// SIMATIC S7-200 project (STEP 7-Micro/WIN), CPU 226 REL 02.00

SYMBOL_TABLE I
                 ?0_40_0  // 镀镍反应池加碱压力开关71
                 ?0_40_0  // 配碱切断阀
                 ?0_40_0  // 配酸切断阀
PDT101           AIW0     // PDT101（镀镍废水过滤器）
AIT101           AIW2     // AIT101PH（镀镍废水调节池PH）
AIT102           AIW4     // AIT102PH（镀镍反应池1#PH）
AIT103           AIW6     // AIT103PH（镀镍反应池2#PH）
FIQ100           AIW8     // FIQ100（镀镍进水总计量）
LT401            AIW10    // 酸液位LT401
LT402            AIW12    // 碱液位LT402
                 AIW14    // 可燃气体报警（未找到）
AIT106           AIW16    // AIT106（NF进水CI）
LS101A           I0.0     // 1#中继池液位高
LS101B           I0.1     // 1#中继池液位高高
M103C_RUN        I0.3     // 反应池搅拌机A运行反馈
M101A_RUN        I0.4     // 镀镍1#中继池提升泵A运行反馈
M101B_RUN        I0.5     // 镀镍1#中继池提升泵B运行反馈
M103D_RUN        I0.6     // 反应池搅拌机B运行反馈
M103C_OVER       I0.7     // 反应池搅拌机A过载
M101A_OVER       I1.0     // 镀镍1#中继池泵A运行过载
M101B_OVER       I1.1     // 镀镍1#中继池泵B运行过载
M103D_OVER       I1.2     // 反应池搅拌机B过载
DUNIE2_H         I1.3     // 镀镍2#中继池液位高
YJC_1A_RUN       I1.4     // 1#应急池提升泵A运行状态14
YJC_1B_RUN       I1.5     // 1#应急池提升泵B运行状态15
YJC_2A_RUN       I1.6     // 2#应急池提升泵A运行状态16
YJC_2B_RUN       I1.7     // 2#应急池提升泵B运行状态17
M402A_RUN        I2.0     // 碱泵A运行反馈M401C
M402B_RUN        I2.1     // 碱泵B运行反馈M401D
M401A_RUN        I2.2     // 酸泵A运行反馈M401A
M401B_RUN        I2.3     // 酸泵B运行反馈M401B
YJC_1A_OVER      I2.4     // 1#应急池提升泵A过载状态24
YJC_1B_OVER      I2.5     // 1#应急池提升泵B过载状态25
YJC_1L           I2.6     // 1#应急池液位计低2.6
YJC_1H           I2.7     // 1#应急池液位计高2.7
YJC_2L           I3.0     // 2#应急池液位计低3.0
YJC_2H           I3.1     // 2#应急池液位计高3.1
JIAN_YEWEI       I3.2     // 镀镍反应池加碱液位计no
DUNIE2_L         I3.3     // 镀镍2#中继池液位低
YJC_2A_OVER      I3.4     // 2#应急池提升泵A过载状态34
YJC_2B_OVER      I3.5     // 2#应急池提升泵B过载状态35
M402A_OVER       I3.6     // 碱泵A过载M401C
M402B_OVER       I3.7     // 碱泵B过载M401D
M401A_OVER       I4.0     // 酸泵A过载M401A
M401B_OVER       I4.1     // 酸泵B过载M401B
JBJ_QPJ_RUN      I5.0     // 配消泡剂搅拌机运行状态60
M410_OVER        I5.1     // 配PAC搅拌机过载状态61
M103E_OVER       I5.2     // 镀镍反应池加碱过载状态62
M401C_OVER       I5.3     // 配酸搅拌机过载状态63
M402C_OVER       I5.4     // 配碱搅拌机过载状态64
JBJ_QPJ_OVER     I5.5     // 配消泡剂搅拌机过载状态65
M410_RUN         I6.4     // 配PAC搅拌机运行状态54
M103E_RUN        I6.5     // 镀镍反应池加碱运行状态55
M401C_RUN        I6.6     // 配酸搅拌机运行状态56
M402C_RUN        I6.7     // 配碱搅拌机运行状态57
UF_YW_H          I7.0     // 超滤中间水箱液位高
SV106A_RUN       I7.1     // 过滤器切断阀1运行反馈
SV106B_RUN       I7.2     // 过滤器切断阀2运行反馈
SV106C_RUN       I7.3     // 过滤器切断阀3运行反馈
DUNIE_A_RUN      I7.4     // 镀镍2#中继池提升泵B运行
DUNIE_B_RUN      I7.5     // 镀镍2#中继池提升泵A运行
DUNIE_A_OVER     I7.6     // 镀镍2#中继池提升泵B过载
DUNIE_B_OVER     I7.7     // 镀镍2#中继池提升泵A过载
M103A_RUN        I8.2     // 镀镍调节池提升泵A运行状态82
M103B_RUN        I8.3     // 镀镍调节池提升泵B运行状态83
M103A_OVER       I8.4     // 镀镍调节池提升泵A过载状态84
M103B_OVER       I8.5     // 镀镍调节池提升泵B过载状态85
TJCYW_L          I8.6     // 镀镍调节池液位计(起泵位)8.6
TJCYW_H          I8.7     // 镀镍调节池液位计(低保护)8.7
                          // 集水井液位计no
END_SYMBOL_TABLE

SYMBOL_TABLE Q
                 ?0_40_0  // 集水井提升泵A运行
                 ?0_40_0  // 集水井提升泵B运行
M101A            Q0.0     // 镀镍1#中继池提升泵A运行00
M101B            Q0.1     // 镀镍1#中继池提升泵B运行01
DUNIE_A          Q0.2     // 镀镍2#中继池提升泵B运行7#
DUNIE_B          Q0.3     // 镀镍2#中继池提升泵A运行7#
YJC_PUMPA        Q0.4     // 应急池提升泵A
YJC_PUMPB        Q0.5     // 应急池提升泵B
YJC_PUMPC        Q0.6     // 应急池提升泵C
YJC_PUMPD        Q0.7     // 应急池提升泵D
M402A            Q1.0     // 酸提升泵A
M402B            Q1.1     // 酸提升泵B
M401A            Q1.2     // 碱提升泵A
M401B            Q1.3     // 碱提升泵B
M410             Q2.1     // 配PAC搅拌机运行54
M103E            Q2.2     // 镀镍反应池加碱运行22
M401C            Q2.3     // 配酸搅拌机运行23
M402C            Q2.4     // 配碱搅拌机运行57
JBJ_QPJ          Q2.5     // 配消泡剂搅拌机运行60
LV401            Q2.6     // 酸加水阀门26
LV402            Q2.7     // 碱加水阀门27
M103A            Q3.0     // 镀镍调节池池提升泵A
M103B            Q3.1     // 镀镍调节池池提升泵B
M103C            Q3.2     // 反应池搅拌机Ano
M103D            Q3.3     // 反应池搅拌机Bno
SV106A           Q3.4     // 过滤器切断阀1no
SV106B           Q3.5     // 过滤器切断阀2no
SV106C           Q3.6     // 过滤器切断阀3no
END_SYMBOL_TABLE

SYMBOL_TABLE M
AUTO             M0.0     // 手/自动
                 M0.2     // 中间水箱液位高标志
                 M0.3     // 调节池泵启动条件
                 M0.4     // M401AB
                 M0.5     // M402AB
SV106_ID         M0.7     // 置过滤器截断阀运行标志位
                 M1.0     // 镀镍2#中继池启动条件
                 M1.1     // 1#应急池提升泵启动条件
                 M1.2     // 2#应急池提升泵启动条件
                 M1.3     // 镀镍1#中继池启动条件
FYC_ALARM        M1.4     // 反应池PH报警
ALARM_EN         M2.0     // 报警
TJC_ALARM        M2.1     // 调节池PH报警
TJC_ALARM_R      M2.2     // 调节池PH报警复位
                 M10.0    // AIT101报警
                 M10.1    // PDT101报警
                 M10.2    // AIT102报警
                 M10.3    // AIT103报警
                 M10.4    // FE101报警
                 M10.5    // 可燃气体报警
                 M10.6    // 酸液位报警
                 M10.7    // 碱液位报警
                 M11.0    // AIT106报警
M112             M11.2    // 镀镍2#中继池提升泵A在线
M113             M11.3    // 镀镍2#中继池提升泵B在线
M156             M15.6    // 酸单次配药
M157             M15.7    // 碱单次配药
M160             M16.0    // 反应池PH压力联锁允许
M161             M16.1    // 反应池PH液位联锁允许
M162             M16.2    // 反应池PH自动控制
M163             M16.3    // 调节池提升泵允许PH控制
M164             M16.4    // 调节池PH报警
M165             M16.5    // 过滤器压力报警允许
M166             M16.6    // 调节池液位允许提升泵启动综合状态
M167             M16.7    // 酸自动配药
M170             M17.0    // 碱自动配药
M171             M17.1    // 2#应急池提升泵液位联锁允许
M172             M17.2    // 1#应急池提升泵液位联锁允许
M173             M17.3    // 镀镍调节池提升泵液位联锁允许
M174             M17.4    // 镀镍2#中继池提升泵液位联锁允许
M175             M17.5    // 镀镍1#中继池提升泵液位联锁允许
M176             M17.6    // 镀镍反应池搅拌机联锁允许
M182             M18.2    // 集水井提升泵B在线
M183             M18.3    // 集水井提升泵A在线
M184             M18.4    // 配消泡剂搅拌机在线
M185             M18.5    // 配PAC搅拌机在线
M186             M18.6    // 配碱搅拌机在线
M187             M18.7    // 配酸搅拌机在线
M190             M19.0    // 碱输送泵A在线
M191             M19.1    // 碱输送泵B在线
M192             M19.2    // 酸输送泵A在线
M193             M19.3    // 酸输送泵B在线
M194             M19.4    // 2#应急池提升泵B在线
M195             M19.5    // 2#应急池提升泵A在线
M196             M19.6    // 1#应急池提升泵B在线
M197             M19.7    // 1#应急池提升泵A在线
M200             M20.0    // 镀镍反应池加碱在线
M201             M20.1    // 镀镍反应池搅拌机A在线
M202             M20.2    // 镀镍反应池搅拌机B在线
M203             M20.3    // 镀镍调节池提升泵A在线
M204             M20.4    // 镀镍调节池提升泵B在线
M205             M20.5    // 镀镍1#中继池提升泵A在线
M206             M20.6    // 镀镍1#中继池提升泵B在线
M211             M21.1    // 过滤器切断阀1在线
M212             M21.2    // 过滤器切断阀2在线
M213             M21.3    // 过滤器切断阀3在线
M214             M21.4    // 镀镍反应池加碱压力保护允许
M215             M21.5    // 过滤器切断阀
END_SYMBOL_TABLE

SYMBOL_TABLE TC
                 T37      // AB切换定时
                 T38      // AB定时辅助
                 T254     // 报警延时
END_SYMBOL_TABLE

SYMBOL_TABLE V
                 VD300    // AIT101最大设定值
                 VD304    // AIT101最小设定值
                 VD308    // PDT101最大设定值
                 VD312    // PDT101最小设定值
                 VD316    // AIT102最大设定值
                 VD320    // AIT102最小设定值
                 VD324    // AIT103最大设定值
                 VD328    // AIT103最小设定值
                 VD332    // FE101最大设定值
                 VD336    // FE101最小设定值
                 VD340    // 可燃气体报警最大设定值
                 VD344    // 可燃气体报警最小设定值
                 VD348    // 酸液位最大设定值
                 VD352    // 酸液位最小设定值
                 VD356    // 碱液位最大设定值
                 VD360    // 碱液位最小设定值
                 VD364    // AIT106最大设定值
                 VD368    // AIT106最小设定值
PDT              VW0      // PDT101
TJC_PH           VW2      // AIT101
FYC_PH1          VW4      // AIT102
FYC_PH2          VW6      // AIT103
FE101            VW8      // FE101
SUAN_YW          VW10     // 酸液位
JIAN_YW          VW12     // 碱液位
                 VW14     // 可燃气体报警
                 VW16     // AIT106镀镍纳虑进水电导率
S125             VW18     // 调节池PH报警设定值高8.0
S126             VW20     // 反应池PH1低限设定值6.0
S127             VW22     // 反应池PH1高限设定值8.0
S128             VW24     // 酸加水高度设定值1-30
S129             VW26     // 酸加酸高度设定值2-60
S130             VW28     // 酸加水高度设定值3-100
S131             VW30     // 碱加水高度设定值1
S132             VW32     // 碱加碱高度设定值2
S133             VW34     // 碱加水高度设定值3
                 VW36     // 调节池PH报警设定值低
                 VW42     // PDT101最大设定值10
TIME1            VW100    // 定时切换时间(分钟)30
END_SYMBOL_TABLE

ORGANIZATION_BLOCK MAIN:OB1
TITLE=PROGRAM COMMENTS
BEGIN
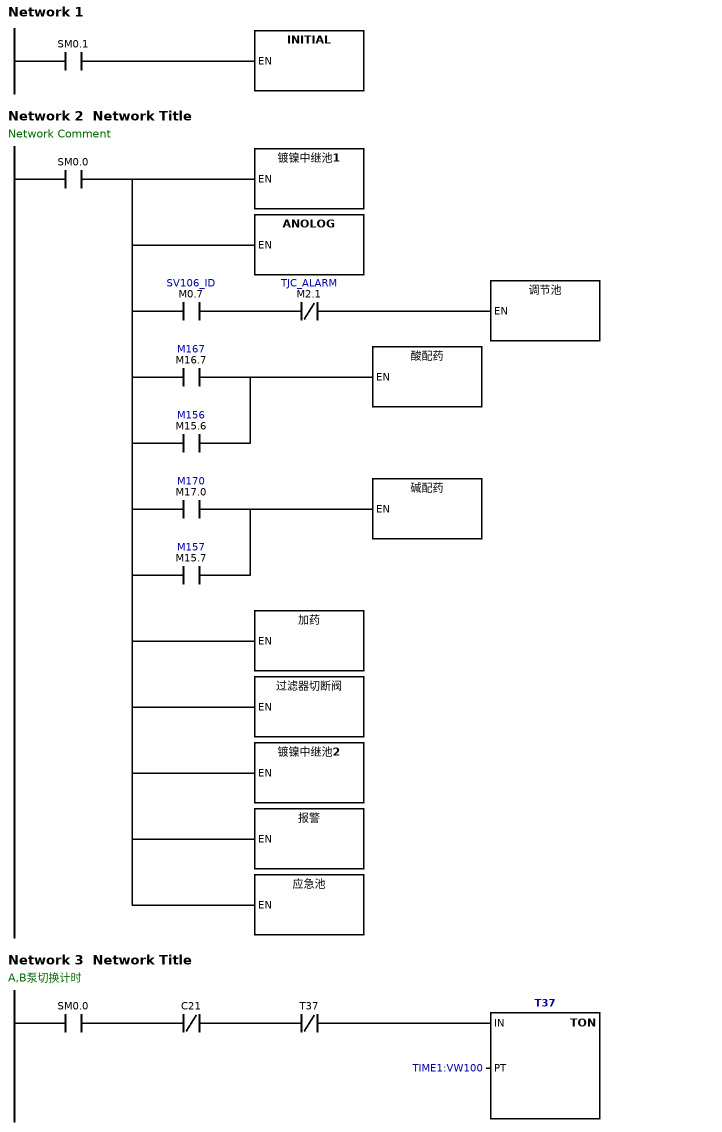
Network 1
// (network saved uncompiled; LAD cells follow)
// row 0: c0 -| |- SM0.1  c1 --  c2 [INITIAL EN:=power@row0]
Network 2 // Network Title
// Network Comment
LD     SM0.0
LPS
CALL   镀镍中继池1:SBR0
CALL   ANOLOG:SBR4
A      SV106_ID:M0.7
AN     TJC_ALARM:M2.1
CALL   调节池:SBR3
LRD
LD     M167:M16.7
O      M156:M15.6
ALD
CALL   酸配药:SBR5
LRD
LD     M170:M17.0
O      M157:M15.7
ALD
CALL   碱配药:SBR6
LPP
CALL   加药:SBR2
CALL   过滤器切断阀:SBR9
CALL   镀镍中继池2:SBR7
CALL   报警:SBR8
CALL   应急池:SBR1
Network 3 // Network Title
// A,B泵切换计时
LD     SM0.0
AN     C21
AN     T37
TON    T37, TIME1:VW100
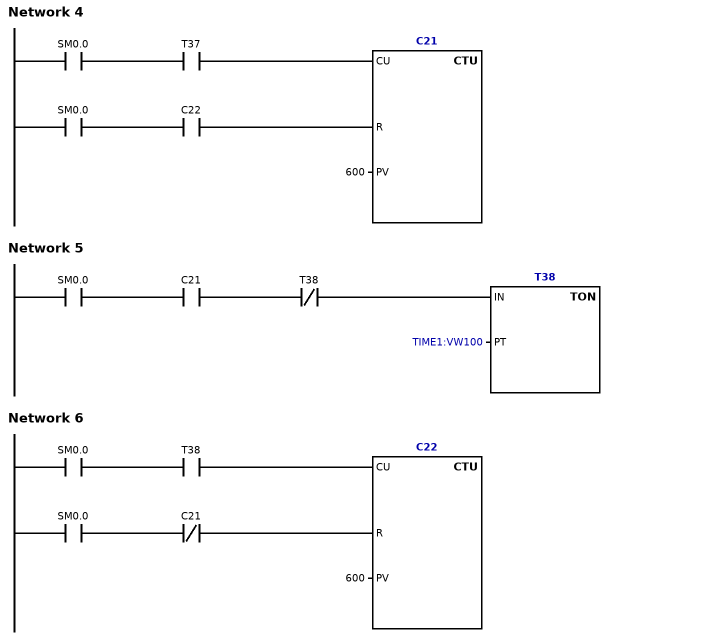
Network 4
LD     SM0.0
A      T37
LD     SM0.0
A      C22
CTU    C21, 600
Network 5
LD     SM0.0
A      C21
AN     T38
TON    T38, TIME1:VW100
Network 6
LD     SM0.0
A      T38
LD     SM0.0
AN     C21
CTU    C22, 600
END_ORGANIZATION_BLOCK

SUBROUTINE_BLOCK 镀镍中继池1:SBR0
TITLE=1#中继池
BEGIN
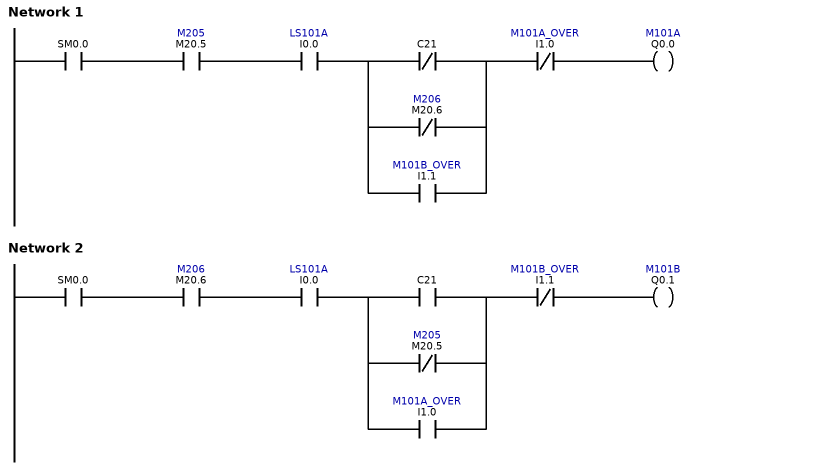
Network 1
LD     SM0.0
A      M205:M20.5
A      LS101A:I0.0
LDN    C21
ON     M206:M20.6
O      M101B_OVER:I1.1
ALD
AN     M101A_OVER:I1.0
=      M101A:Q0.0
Network 2
LD     SM0.0
A      M206:M20.6
A      LS101A:I0.0
LD     C21
ON     M205:M20.5
O      M101A_OVER:I1.0
ALD
AN     M101B_OVER:I1.1
=      M101B:Q0.1
END_SUBROUTINE_BLOCK

SUBROUTINE_BLOCK 应急池:SBR1
TITLE=子程序注释
BEGIN
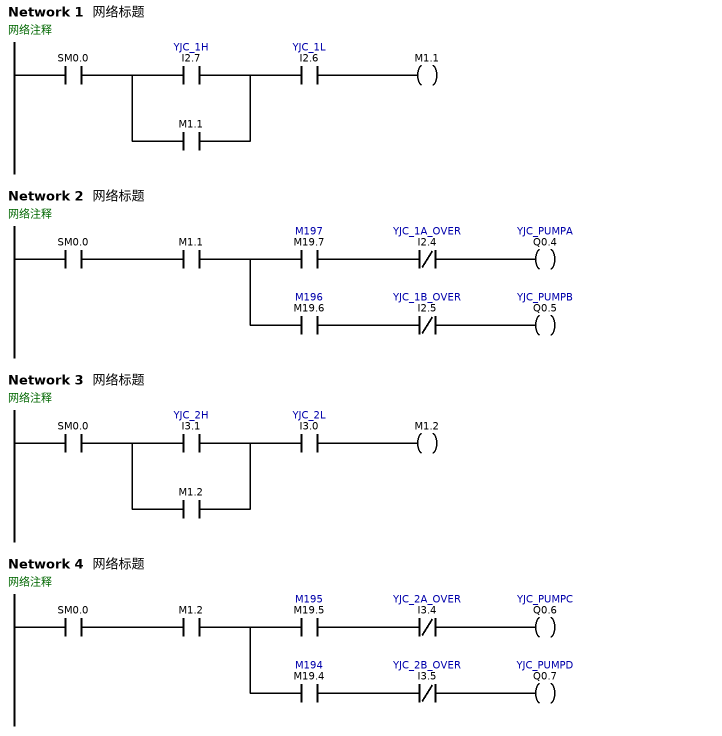
Network 1 // 网络标题
// 网络注释
LD     SM0.0
LD     YJC_1H:I2.7
O      M1.1
ALD
A      YJC_1L:I2.6
=      M1.1
Network 2 // 网络标题
// 网络注释
LD     SM0.0
A      M1.1
LPS
A      M197:M19.7
AN     YJC_1A_OVER:I2.4
=      YJC_PUMPA:Q0.4
LPP
A      M196:M19.6
AN     YJC_1B_OVER:I2.5
=      YJC_PUMPB:Q0.5
Network 3 // 网络标题
// 网络注释
LD     SM0.0
LD     YJC_2H:I3.1
O      M1.2
ALD
A      YJC_2L:I3.0
=      M1.2
Network 4 // 网络标题
// 网络注释
LD     SM0.0
A      M1.2
LPS
A      M195:M19.5
AN     YJC_2A_OVER:I3.4
=      YJC_PUMPC:Q0.6
LPP
A      M194:M19.4
AN     YJC_2B_OVER:I3.5
=      YJC_PUMPD:Q0.7
END_SUBROUTINE_BLOCK

SUBROUTINE_BLOCK 加药:SBR2
TITLE=各加药泵
BEGIN
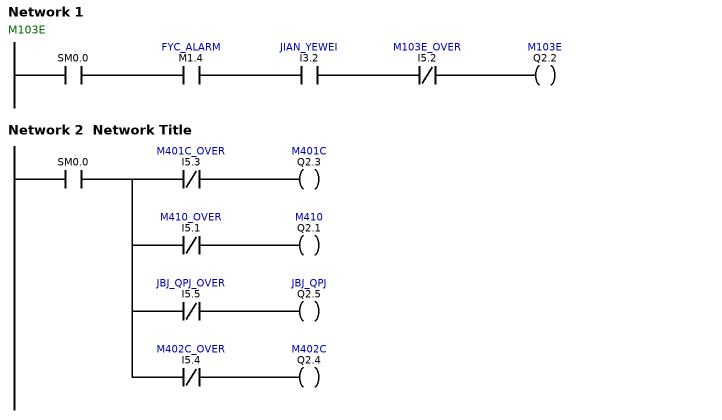
Network 1
// M103E
LD     SM0.0
A      FYC_ALARM:M1.4
A      JIAN_YEWEI:I3.2
AN     M103E_OVER:I5.2
=      M103E:Q2.2
Network 2 // Network Title
LD     SM0.0
LPS
AN     M401C_OVER:I5.3
=      M401C:Q2.3
LRD
AN     M410_OVER:I5.1
=      M410:Q2.1
LRD
AN     JBJ_QPJ_OVER:I5.5
=      JBJ_QPJ:Q2.5
LPP
AN     M402C_OVER:I5.4
=      M402C:Q2.4
END_SUBROUTINE_BLOCK

SUBROUTINE_BLOCK 调节池:SBR3
TITLE=调节池
BEGIN
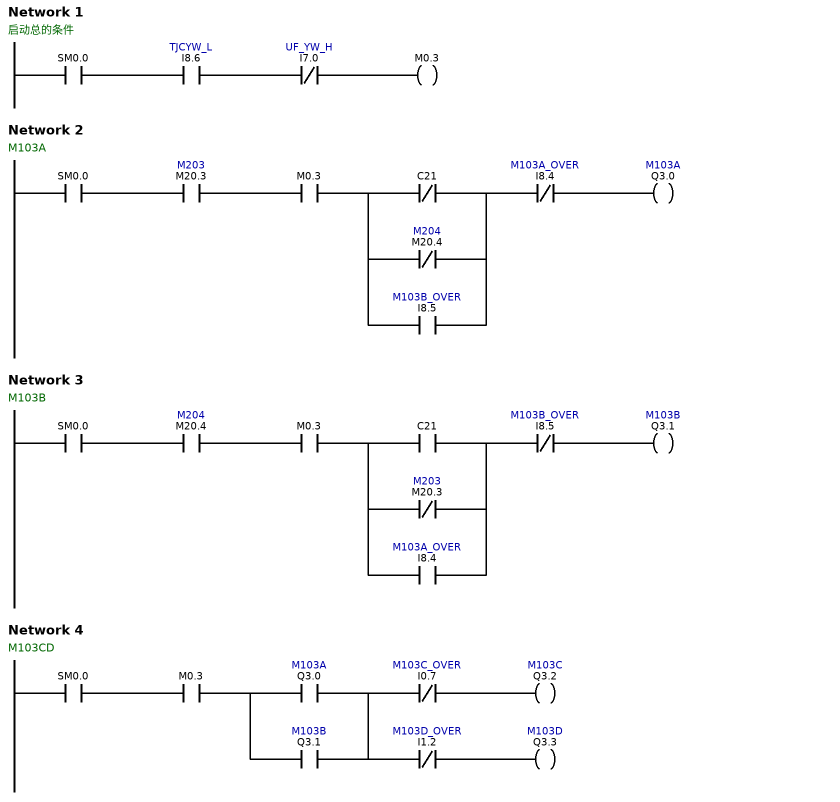
Network 1
// 启动总的条件
LD     SM0.0
A      TJCYW_L:I8.6
AN     UF_YW_H:I7.0
=      M0.3
Network 2
// M103A
LD     SM0.0
A      M203:M20.3
A      M0.3
LDN    C21
ON     M204:M20.4
O      M103B_OVER:I8.5
ALD
AN     M103A_OVER:I8.4
=      M103A:Q3.0
Network 3
// M103B
LD     SM0.0
A      M204:M20.4
A      M0.3
LD     C21
ON     M203:M20.3
O      M103A_OVER:I8.4
ALD
AN     M103B_OVER:I8.5
=      M103B:Q3.1
Network 4
// M103CD
LD     SM0.0
A      M0.3
LD     M103A:Q3.0
O      M103B:Q3.1
ALD
LPS
AN     M103C_OVER:I0.7
=      M103C:Q3.2
LPP
AN     M103D_OVER:I1.2
=      M103D:Q3.3
END_SUBROUTINE_BLOCK

SUBROUTINE_BLOCK ANOLOG:SBR4
TITLE=SUBROUTINE COMMENTS
BEGIN
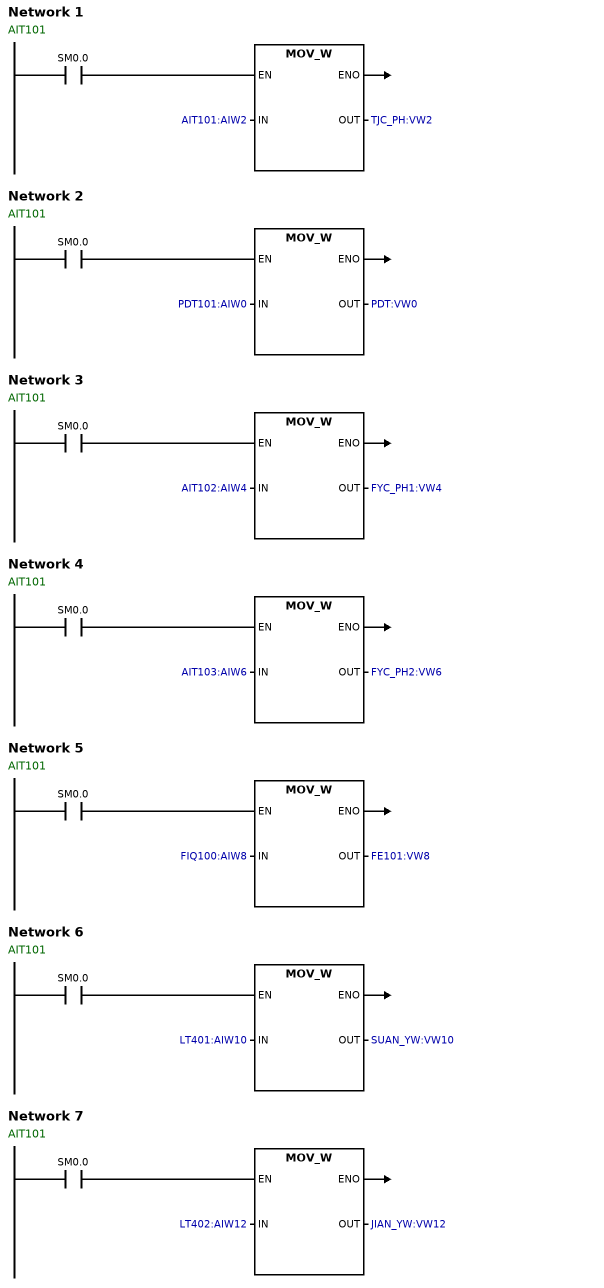
Network 1
// AIT101
LD     SM0.0
MOVW   AIT101:AIW2, TJC_PH:VW2
Network 2
// AIT101
LD     SM0.0
MOVW   PDT101:AIW0, PDT:VW0
Network 3
// AIT101
LD     SM0.0
MOVW   AIT102:AIW4, FYC_PH1:VW4
Network 4
// AIT101
LD     SM0.0
MOVW   AIT103:AIW6, FYC_PH2:VW6
Network 5
// AIT101
LD     SM0.0
MOVW   FIQ100:AIW8, FE101:VW8
Network 6
// AIT101
LD     SM0.0
MOVW   LT401:AIW10, SUAN_YW:VW10
Network 7
// AIT101
LD     SM0.0
MOVW   LT402:AIW12, JIAN_YW:VW12
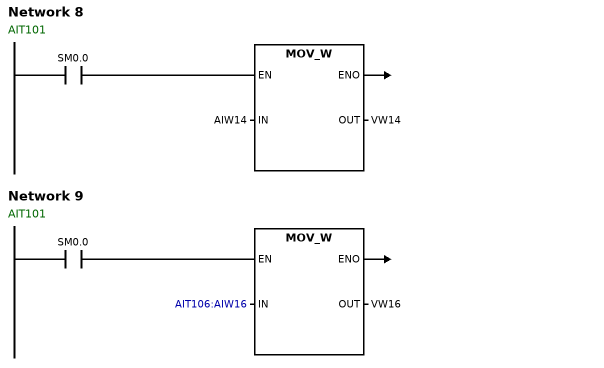
Network 8
// AIT101
LD     SM0.0
MOVW   AIW14, VW14
Network 9
// AIT101
LD     SM0.0
MOVW   AIT106:AIW16, VW16
END_SUBROUTINE_BLOCK

SUBROUTINE_BLOCK 酸配药:SBR5
TITLE=
BEGIN
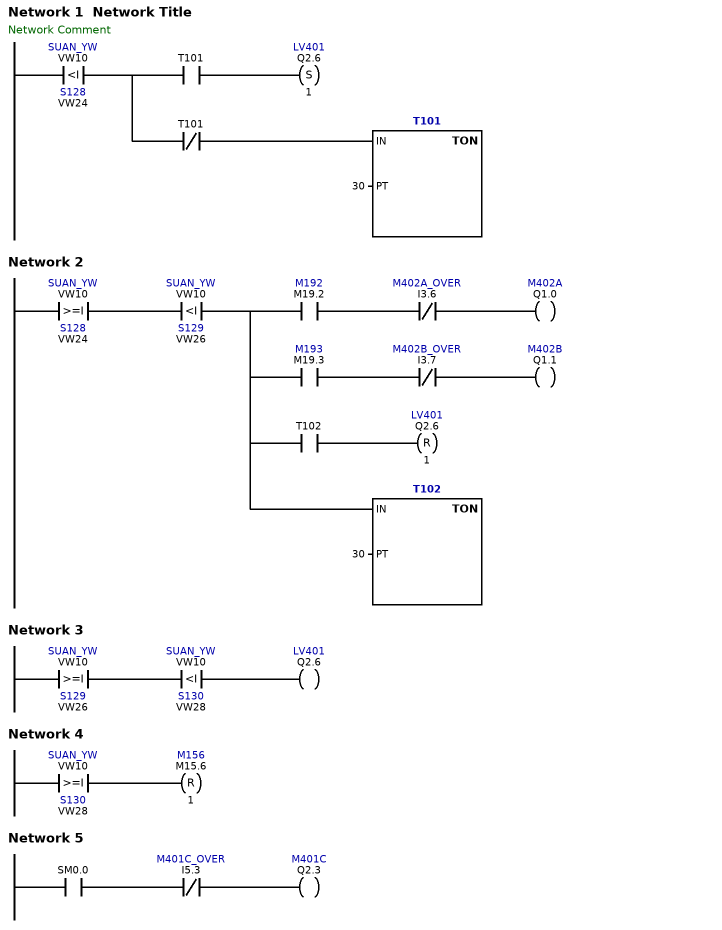
Network 1 // Network Title
// Network Comment
LDW<   SUAN_YW:VW10, S128:VW24
LPS
A      T101
S      LV401:Q2.6, 1
LPP
AN     T101
TON    T101, 30
Network 2
LDW>=  SUAN_YW:VW10, S128:VW24
AW<    SUAN_YW:VW10, S129:VW26
LPS
A      M192:M19.2
AN     M402A_OVER:I3.6
=      M402A:Q1.0
LRD
A      M193:M19.3
AN     M402B_OVER:I3.7
=      M402B:Q1.1
LRD
A      T102
R      LV401:Q2.6, 1
LPP
TON    T102, 30
Network 3
LDW>=  SUAN_YW:VW10, S129:VW26
AW<    SUAN_YW:VW10, S130:VW28
=      LV401:Q2.6
Network 4
LDW>=  SUAN_YW:VW10, S130:VW28
R      M156:M15.6, 1
Network 5
LD     SM0.0
AN     M401C_OVER:I5.3
=      M401C:Q2.3
END_SUBROUTINE_BLOCK

SUBROUTINE_BLOCK 碱配药:SBR6
TITLE=
BEGIN
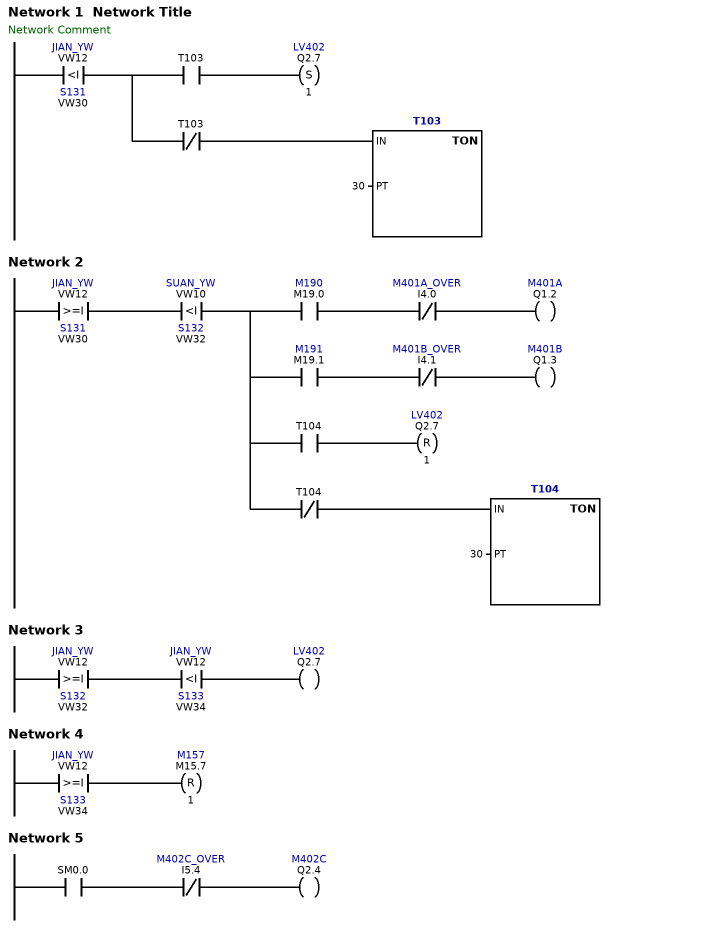
Network 1 // Network Title
// Network Comment
LDW<   JIAN_YW:VW12, S131:VW30
LPS
A      T103
S      LV402:Q2.7, 1
LPP
AN     T103
TON    T103, 30
Network 2
LDW>=  JIAN_YW:VW12, S131:VW30
AW<    SUAN_YW:VW10, S132:VW32
LPS
A      M190:M19.0
AN     M401A_OVER:I4.0
=      M401A:Q1.2
LRD
A      M191:M19.1
AN     M401B_OVER:I4.1
=      M401B:Q1.3
LRD
A      T104
R      LV402:Q2.7, 1
LPP
AN     T104
TON    T104, 30
Network 3
LDW>=  JIAN_YW:VW12, S132:VW32
AW<    JIAN_YW:VW12, S133:VW34
=      LV402:Q2.7
Network 4
LDW>=  JIAN_YW:VW12, S133:VW34
R      M157:M15.7, 1
Network 5
LD     SM0.0
AN     M402C_OVER:I5.4
=      M402C:Q2.4
END_SUBROUTINE_BLOCK

SUBROUTINE_BLOCK 镀镍中继池2:SBR7
TITLE=
BEGIN
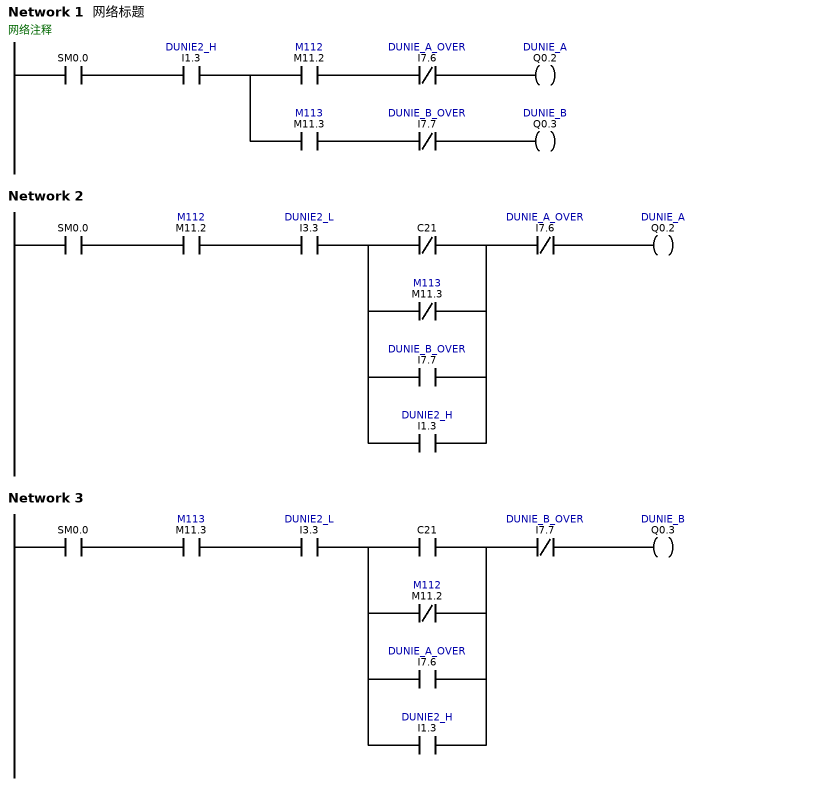
Network 1 // 网络标题
// 网络注释
LD     SM0.0
A      DUNIE2_H:I1.3
LPS
A      M112:M11.2
AN     DUNIE_A_OVER:I7.6
=      DUNIE_A:Q0.2
LPP
A      M113:M11.3
AN     DUNIE_B_OVER:I7.7
=      DUNIE_B:Q0.3
Network 2
LD     SM0.0
A      M112:M11.2
A      DUNIE2_L:I3.3
LDN    C21
ON     M113:M11.3
O      DUNIE_B_OVER:I7.7
O      DUNIE2_H:I1.3
ALD
AN     DUNIE_A_OVER:I7.6
=      DUNIE_A:Q0.2
Network 3
LD     SM0.0
A      M113:M11.3
A      DUNIE2_L:I3.3
LD     C21
ON     M112:M11.2
O      DUNIE_A_OVER:I7.6
O      DUNIE2_H:I1.3
ALD
AN     DUNIE_B_OVER:I7.7
=      DUNIE_B:Q0.3
END_SUBROUTINE_BLOCK

SUBROUTINE_BLOCK 报警:SBR8
TITLE=子程序注释
BEGIN
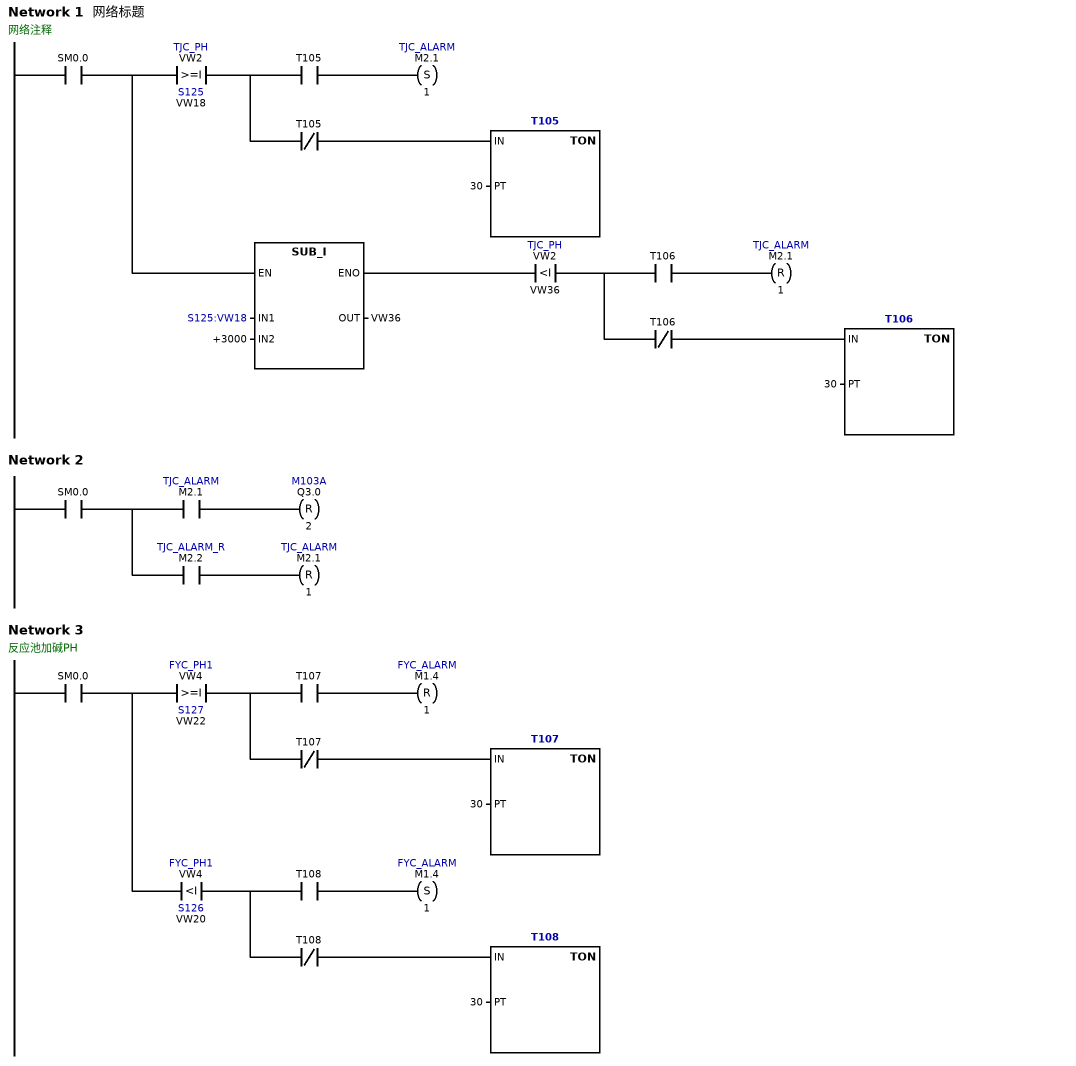
Network 1 // 网络标题
// 网络注释
LD     SM0.0
LPS
AW>=   TJC_PH:VW2, S125:VW18
LPS
A      T105
S      TJC_ALARM:M2.1, 1
LPP
AN     T105
TON    T105, 30
LPP
MOVW   S125:VW18, VW36
AENO
-I     +3000, VW36
AENO
AW<    TJC_PH:VW2, VW36
LPS
A      T106
R      TJC_ALARM:M2.1, 1
LPP
AN     T106
TON    T106, 30
Network 2
LD     SM0.0
LPS
A      TJC_ALARM:M2.1
R      M103A:Q3.0, 2
LPP
A      TJC_ALARM_R:M2.2
R      TJC_ALARM:M2.1, 1
Network 3
// 反应池加碱PH
LD     SM0.0
LPS
AW>=   FYC_PH1:VW4, S127:VW22
LPS
A      T107
R      FYC_ALARM:M1.4, 1
LPP
AN     T107
TON    T107, 30
LPP
AW<    FYC_PH1:VW4, S126:VW20
LPS
A      T108
S      FYC_ALARM:M1.4, 1
LPP
AN     T108
TON    T108, 30
END_SUBROUTINE_BLOCK

SUBROUTINE_BLOCK 过滤器切断阀:SBR9
TITLE=
BEGIN
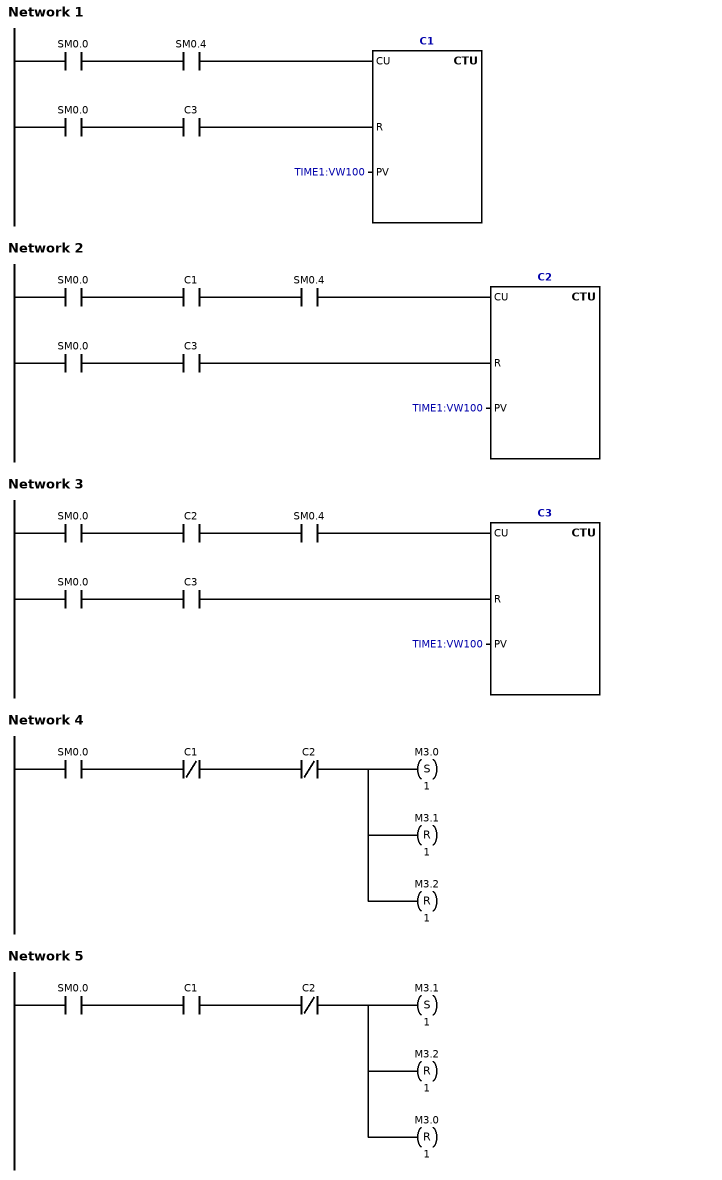
Network 1
LD     SM0.0
A      SM0.4
LD     SM0.0
A      C3
CTU    C1, TIME1:VW100
Network 2
LD     SM0.0
A      C1
A      SM0.4
LD     SM0.0
A      C3
CTU    C2, TIME1:VW100
Network 3
LD     SM0.0
A      C2
A      SM0.4
LD     SM0.0
A      C3
CTU    C3, TIME1:VW100
Network 4
LD     SM0.0
AN     C1
AN     C2
S      M3.0, 1
R      M3.1, 1
R      M3.2, 1
Network 5
LD     SM0.0
A      C1
AN     C2
S      M3.1, 1
R      M3.2, 1
R      M3.0, 1
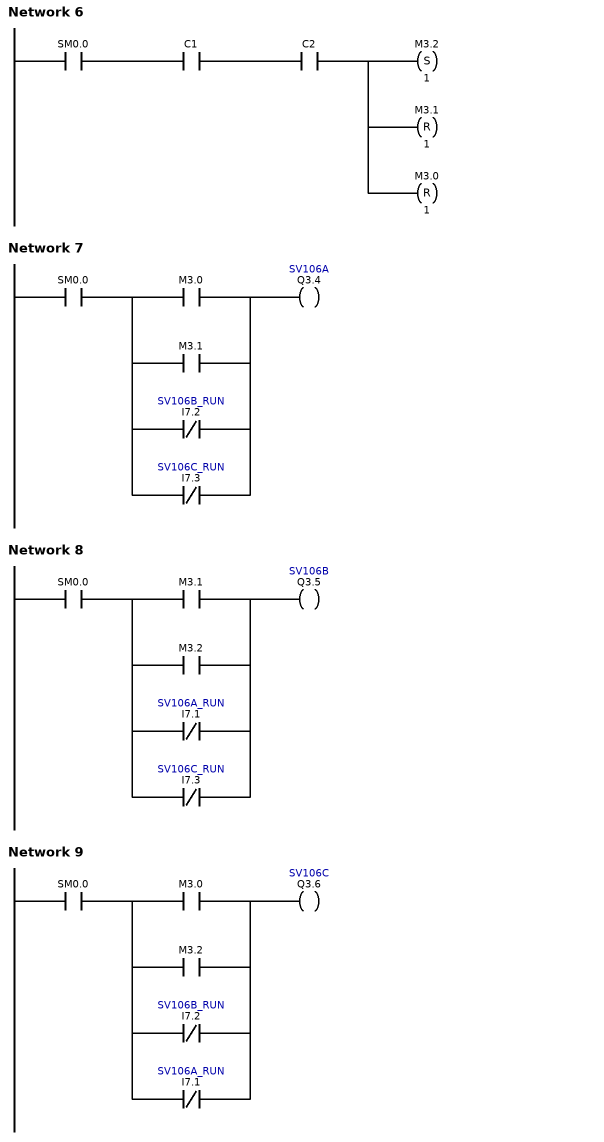
Network 6
LD     SM0.0
A      C1
A      C2
S      M3.2, 1
R      M3.1, 1
R      M3.0, 1
Network 7
LD     SM0.0
LD     M3.0
O      M3.1
ON     SV106B_RUN:I7.2
ON     SV106C_RUN:I7.3
ALD
=      SV106A:Q3.4
Network 8
LD     SM0.0
LD     M3.1
O      M3.2
ON     SV106A_RUN:I7.1
ON     SV106C_RUN:I7.3
ALD
=      SV106B:Q3.5
Network 9
LD     SM0.0
LD     M3.0
O      M3.2
ON     SV106B_RUN:I7.2
ON     SV106A_RUN:I7.1
ALD
=      SV106C:Q3.6
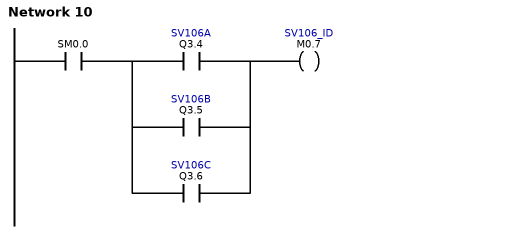
Network 10
LD     SM0.0
LD     SV106A:Q3.4
O      SV106B:Q3.5
O      SV106C:Q3.6
ALD
=      SV106_ID:M0.7
END_SUBROUTINE_BLOCK

SUBROUTINE_BLOCK INITIAL:SBR10
TITLE=子程序注释
BEGIN
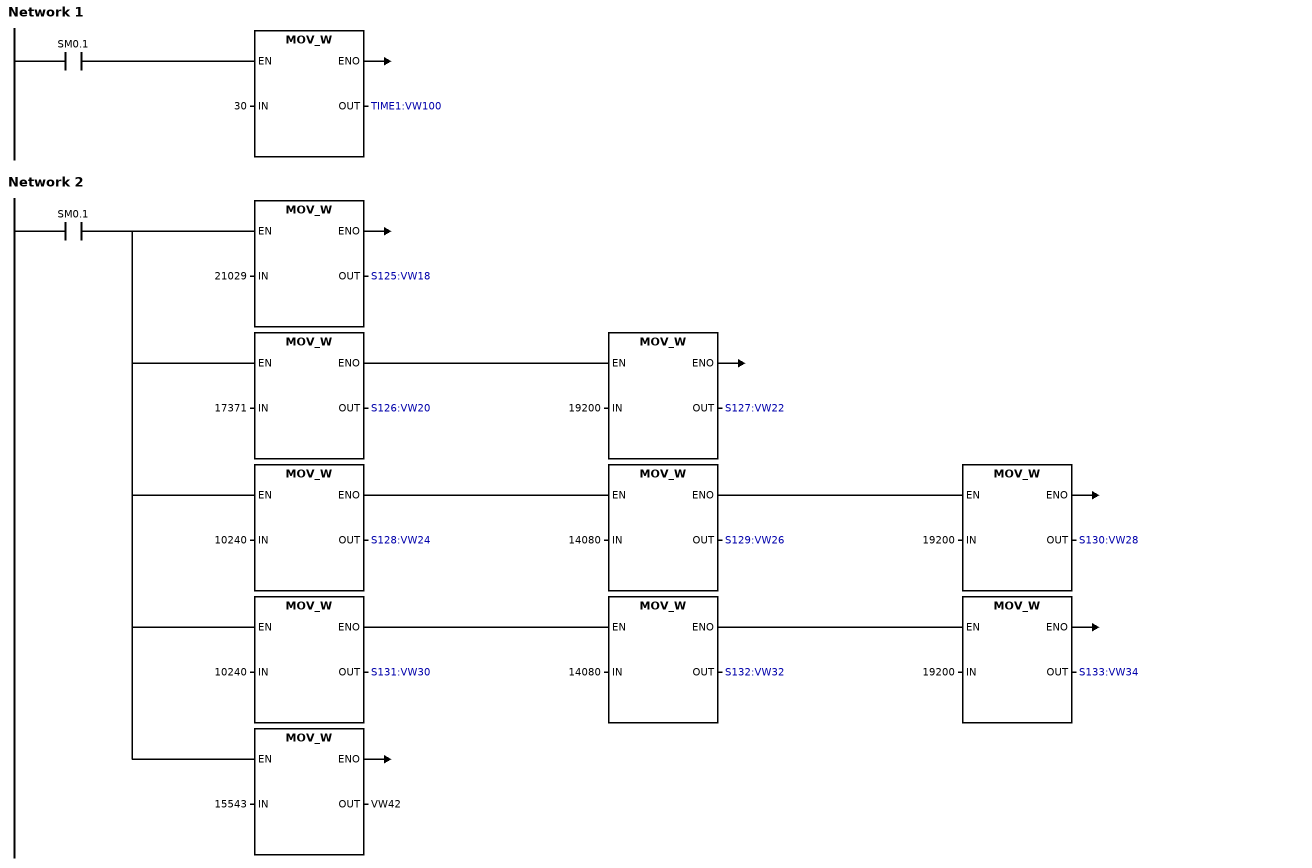
Network 1
LD     SM0.1
MOVW   30, TIME1:VW100
Network 2
LD     SM0.1
LPS
MOVW   21029, S125:VW18
MOVW   17371, S126:VW20
AENO
MOVW   19200, S127:VW22
LRD
MOVW   10240, S128:VW24
AENO
MOVW   14080, S129:VW26
AENO
MOVW   19200, S130:VW28
LRD
MOVW   10240, S131:VW30
AENO
MOVW   14080, S132:VW32
AENO
MOVW   19200, S133:VW34
LPP
MOVW   15543, VW42
END_SUBROUTINE_BLOCK
